FUNCTION_BLOCK E_MUX_4 (* Event multiplexer (generic FB) *)
  (* Standard: 61499-1 Annex A; Description: Copyright (c) 2017, 2025 fortiss GmbH, HR Agrartechnik GmbH This program and the accompanying materials are made available under the terms of the Eclipse Public License 2.0 which is available at https://www.eclipse.org/legal/epl-2.0/ SPDX-License-Identifier: EPL-2.0 *)
  (* Version 1.0, 2017-09-22, Alois Zoitl, fortiss GmbH, initial API and implementation and/or initial documentation *)
  (* Version 1.1, 2025-02-16, Franz Höpfinger, HR Agrartechnik GmbH, Copy E_DEMUX and made E_MUX *)
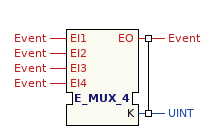
  EVENT_INPUT
    EI1; (* Event to multiplex, K=0 *)
    EI2; (* Event to multiplex, K=1 *)
    EI3; (* Event to multiplex, K=2 *)
    EI4; (* Event to multiplex, K=3 *)
  END_EVENT
  EVENT_OUTPUT
    EO WITH K; (* Event which was multiplexed *)
  END_EVENT
  VAR_OUTPUT
    K : UINT; (* Event index *)
  END_VAR
END_FUNCTION_BLOCK
